FUNCTION TryConvert_BYTE_TO_DWORD : BOOL
VAR_INPUT
	in : BYTE;
	out : REFERENCE TO DWORD;
END_VAR

out := BYTE_TO_DWORD(in);
TryConvert_BYTE_TO_DWORD := TRUE;

END_FUNCTION

(* stored: Version 1.1.0.1, ProductVersion 3.1.4024.12
   POU TryConvert_BYTE_TO_DWORD: Id {3c8d5610-9ac6-4fe9-bf32-e3396a2c6fd9}, SpecialFunc None *)
